Fanuc KAREL source: kb00116.KL

-- PROVISIONAL review KL for V940-1; original PC SHA256 c18feafd0ccbf98bb6a1968d35a668035799b71d0021534fb2101f2ea2bdcc49
-- Incomplete behavior may be omitted. Consult companion uncertainty JSON. Do not deploy.
PROGRAM KB00116
%NOLOCKGROUP
VAR
  P1 : REAL
  RESULT : REAL
BEGIN
  -- V9_ZERO_TABLE_METADATA_HINT layout=0001; no indexed target words; source/name/runtime held
  -- UNRESOLVED_PC offsets 5-16; opcodes 2E,23
  -- UNRESOLVED_PC offsets 21-36; opcodes 27,22,76,23
  -- UNRESOLVED_PC offsets 41-45; opcodes 7F
END KB00116
